FUNCTION_BLOCK MOYENNE
VAR_INPUT
	In_valeur: REAL;
	In_synchro: BOOL;
	In_fenetre_mesure: TIME;
END_VAR
VAR_OUTPUT
	Out_fenetre_mesure: TIME;
	Out_fin: BOOL;
	Out_Moyenne_0: REAL;
	Out_Moyenne_1: REAL;
END_VAR
VAR
	F_Fenetre_mesure_active: F_TRIG;
	R_In_Synchro: R_TRIG;
	TOF_0: TOF;
	Fenetre_mesure_active: BOOL;
	Nbr_valeur_mesure: REAL;
END_VAR

ACTION Calcul:
(* Gestion des fronts montants et front descendants *)

	R_In_Synchro(CLK := In_Synchro);
	F_Fenetre_mesure_active(CLK := Fenetre_mesure_active);

(* Traitements *)

	IF R_In_Synchro.Q THEN  (* Initialisation des valeurs au lancement de la synchronisation *)
	
		Out_fin:=False; 
		Nbr_valeur_mesure:=0.0; (* RAZ nbr de cycle automate *)
	
	END_IF;
	

	TOF_0 (IN := R_In_Synchro.Q,(* Gestion de la fenêtre de mesure  *)
		  PT := In_fenetre_mesure,
		  Q => Fenetre_mesure_active,
		  ET => Out_fenetre_mesure);
	
	IF Fenetre_mesure_active  THEN (* Traitement durant la fenêtre de mesure *) 
		
		Out_Moyenne_0:=(Out_Moyenne_0*Nbr_valeur_mesure+In_valeur)/(Nbr_valeur_mesure+1.0); (* calcul moyenne *)
	
		Nbr_valeur_mesure:=Nbr_valeur_mesure+1.0; (* calcul nbr de cycle automate *)
	
	ELSIF F_Fenetre_mesure_active.Q THEN (* Traitement en fin de fenêtre de mesure *)
	
		Out_fin:=true;
		Out_Moyenne_1:=Out_Moyenne_0; (* Sauvegarde de la moyenne calculée *)
		Out_Moyenne_0:=0.0; (* RAZ moyenne calculée *)
	
	End_if;
END_ACTION

END_FUNCTION_BLOCK

(* stored: Version 1.1.0.1, ProductVersion 3.1.4024.11
   POU MOYENNE: Id {3ef9cc90-b14c-4561-bfe4-799f51310882}, SpecialFunc None
   Action Calcul: Id {a94ee6e4-071b-454a-b023-19351672753b} *)
